// TIA Portal V20 export
// export: Created 2026-04-11T06:02:30.8431655Z, ExportSetting WithDefaults, DisplayName Totally Integrated Automation Portal, DisplayVersion V20, DisplayName TIA Portal Openness, DisplayVersion V20, DisplayName TIA Portal Version Control Interface, DisplayVersion V20, DisplayName STEP 7 Professional, DisplayVersion V20, DisplayName STEP 7 Safety, DisplayVersion V20, DisplayName WinCC Basic/Comfort/Advanced, DisplayVersion V20, DisplayName WinCC Unified, DisplayVersion V20
TYPE "mettlerToledoInd560Udt"
// stored: IsFailsafeCompliant false
   STRUCT
      readMsgSlot { ExternalWritable := 'False'} : Array[1..4] of Struct
         cmdRespons { ExternalWritable := 'False'} : Struct
            FP_1 { ExternalWritable := 'False'} : Bool;
            FP_2 { ExternalWritable := 'False'} : Bool;
            FP_3 { ExternalWritable := 'False'} : Bool;
            FP_4 { ExternalWritable := 'False'} : Bool;
            FP_5 { ExternalWritable := 'False'} : Bool;
            data_integrity { ExternalWritable := 'False'} : Bool;
            cmdAck1 { ExternalWritable := 'False'} : Bool;
            cmdAck2 { ExternalWritable := 'False'} : Bool;
         END_STRUCT;
         reserved { ExternalWritable := 'False'} : Byte;   // volt
         data { ExternalWritable := 'False'} : Real;
         scale_status { ExternalWritable := 'False'} : Struct
            x08_Enter_Key { ExternalWritable := 'False'} : Bool;
            x09_Input_1 { ExternalWritable := 'False'} : Bool;
            x10_Input_2 { ExternalWritable := 'False'} : Bool;
            x11_Input_3 { ExternalWritable := 'False'} : Bool;
            x12_Motion { ExternalWritable := 'False'} : Bool;
            x13_Net_Mode { ExternalWritable := 'False'} : Bool;
            x14_Data_Integrity_2 { ExternalWritable := 'False'} : Bool;
            x15_Data_OK { ExternalWritable := 'False'} : Bool;
            x00_Target_1 { ExternalWritable := 'False'} : Bool;
            x01_Comparator_1 { ExternalWritable := 'False'} : Bool;
            x02_Targe_2 { ExternalWritable := 'False'} : Bool;
            x03_Comparator_2 { ExternalWritable := 'False'} : Bool;
            x04_Target_3 { ExternalWritable := 'False'} : Bool;
            x05_Alway_true { ExternalWritable := 'False'} : Bool;
            x06_TE_bit_1 { ExternalWritable := 'False'} : Bool;
            x07_TE_bit_2 { ExternalWritable := 'False'} : Bool;
         END_STRUCT;
      END_STRUCT;
      writeMsgSlot { ExternalWritable := 'False'} : Array[1..4] of Struct
         cmd { ExternalWritable := 'False'} : UInt;
         data { ExternalWritable := 'False'} : Real;
      END_STRUCT;
      run { ExternalWritable := 'False'} : Struct   // Data calculated from readMsgSlot
         PF { ExternalWritable := 'False'} : Array[1..4] of USInt;   // Floating point input indication
         cmdAck { ExternalWritable := 'False'} : Array[1..4] of USInt;
      END_STRUCT;
      occupiedMsgSlots { ExternalWritable := 'False'} : Array[1..4] of Bool;
      queryDone { ExternalWritable := 'False'} : Struct
         read { ExternalAccessible := 'False'; ExternalVisible := 'False'; ExternalWritable := 'False'} : Bool;
         write { ExternalAccessible := 'False'; ExternalVisible := 'False'; ExternalWritable := 'False'} : Bool;
      END_STRUCT;
   END_STRUCT;
END_TYPE
